_CFC_ (* Continuous Function Chart, elements in execution order *)
#0 MOVE(EN: SCHU_P2_4_RESET_DF_VALUE, SCHU_P2_4_M_MAXSPEED_df)
#1 SCHU_P2_4_M_MAXSPEED <= #0
#2 MOVE(EN: SCHU_P2_4_RESET_DF_VALUE, SCHU_P2_4_M_MINSPEED_df)
#3 SCHU_P2_4_M_MINSPEED <= #2
#4 MOVE(EN: SCHU_P2_4_RESET_DF_VALUE, SCHU_P2_4_YA2_ZADER_RAS_df)
#5 SCHU_P2_4_YA2_ZADER_RAS <= #4
#6 MOVE(EN: SCHU_P2_4_RESET_DF_VALUE, SCHU_P2_4_YA2_UST_RASSOG_df)
#7 SCHU_P2_4_YA2_UST_RASSOG <= #6
#8 MOVE(EN: SCHU_P2_4_RESET_DF_VALUE, SCHU_P2_4_YA2_ZAD_NEISP_df)
#9 SCHU_P2_4_YA2_ZAD_NEISP <= #8
#10 MOVE(EN: SCHU_P2_4_RESET_DF_VALUE, SCHU_P2_4_YA2_ZAD_NAGR_df)
#11 SCHU_P2_4_YA2_ZAD_NAGR <= #10
#12 MOVE(EN: SCHU_P2_4_RESET_DF_VALUE, SCHU_P2_4_YA3_ZADER_OTK_df)
#13 SCHU_P2_4_YA3_ZADER_OTK <= #12
#14 MOVE(EN: SCHU_P2_4_RESET_DF_VALUE, SCHU_P2_4_YA3_ZADER_RAS_df)
#15 SCHU_P2_4_YA3_ZADER_RAS <= #14
#16 MOVE(EN: SCHU_P2_4_RESET_DF_VALUE, SCHU_P2_4_YA3_UST_RAS_POL_df)
#17 SCHU_P2_4_YA3_UST_RAS_POL <= #16
#18 MOVE(EN: SCHU_P2_4_RESET_DF_VALUE, SCHU_P2_4_YA3_UST_RAS_TEMP_df)
#19 SCHU_P2_4_YA3_UST_RAS_TEMP <= #18
#20 MOVE(EN: SCHU_P2_4_RESET_DF_VALUE, SCHU_P2_4_YA4_ZADER_OTK_TEMP_df)
#21 SCHU_P2_4_YA4_ZADER_OTK_TEMP <= #20
#22 MOVE(EN: SCHU_P2_4_RESET_DF_VALUE, SCHU_P2_4_YA4_ZADER_OTK_df)
#23 SCHU_P2_4_YA4_ZADER_OTK <= #22
#24 MOVE(EN: SCHU_P2_4_RESET_DF_VALUE, SCHU_P2_4_YA4_UST_RAS_TEMP_df)
#25 SCHU_P2_4_YA4_UST_RAS_TEMP <= #24
#26 MOVE(EN: SCHU_P2_4_RESET_DF_VALUE, SCHU_P2_4_YA4_UST_RAS_POL_df)
#27 SCHU_P2_4_YA4_UST_RAS_POL <= #26
#28 MOVE(EN: SCHU_P2_4_RESET_DF_VALUE, SCHU_P2_4_YA2_KP_df)
#29 SCHU_P2_4_YA2_KP <= #28
#30 MOVE(EN: SCHU_P2_4_RESET_DF_VALUE, SCHU_P2_4_YA2_TI_df)
#31 SCHU_P2_4_YA2_TI <= #30
#32 MOVE(EN: SCHU_P2_4_RESET_DF_VALUE, SCHU_P2_4_YA2_TV_df)
#33 SCHU_P2_4_YA2_TV <= #32
#34 MOVE(EN: SCHU_P2_4_RESET_DF_VALUE, SCHU_P2_4_YA2_TD_df)
#35 SCHU_P2_4_YA2_TD <= #34
#36 MOVE(EN: SCHU_P2_4_RESET_DF_VALUE, SCHU_P2_4_YA3_KP_df)
#37 SCHU_P2_4_YA3_KP <= #36
#38 MOVE(EN: SCHU_P2_4_RESET_DF_VALUE, SCHU_P2_4_YA3_TI_df)
#39 SCHU_P2_4_YA3_TI <= #38
#40 MOVE(EN: SCHU_P2_4_RESET_DF_VALUE, SCHU_P2_4_YA3_TV_df)
#41 SCHU_P2_4_YA3_TV <= #40
#42 MOVE(EN: SCHU_P2_4_RESET_DF_VALUE, SCHU_P2_4_YA3_TD_df)
#43 SCHU_P2_4_YA3_TD <= #42
#44 MOVE(EN: SCHU_P2_4_RESET_DF_VALUE, SCHU_P2_4_YA4_KP_df)
#45 SCHU_P2_4_YA4_KP <= #44
#46 MOVE(EN: SCHU_P2_4_RESET_DF_VALUE, SCHU_P2_4_YA4_TI_df)
#47 SCHU_P2_4_YA4_TI <= #46
#48 MOVE(EN: SCHU_P2_4_RESET_DF_VALUE, SCHU_P2_4_YA4_TV_df)
#49 SCHU_P2_4_YA4_TV <= #48
#50 MOVE(EN: SCHU_P2_4_RESET_DF_VALUE, SCHU_P2_4_YA4_TD_df)
#51 SCHU_P2_4_YA4_TD <= #50
#52 MOVE(EN: SCHU_P2_4_RESET_DF_VALUE, SCHU_P2_4_PE_KP_df)
#53 SCHU_P2_4_PE_KP <= #52
#54 MOVE(EN: SCHU_P2_4_RESET_DF_VALUE, SCHU_P2_4_PE_TI_df)
#55 SCHU_P2_4_PE_TI <= #54
#56 MOVE(EN: SCHU_P2_4_RESET_DF_VALUE, SCHU_P2_4_PE_TV_df)
#57 SCHU_P2_4_PE_TV <= #56
#58 MOVE(EN: SCHU_P2_4_RESET_DF_VALUE, SCHU_P2_4_PE_TD_df)
#59 SCHU_P2_4_PE_TD <= #58
#60 MOVE(EN: SCHU_P2_4_RESET_DF_VALUE, SCHU_P2_4_PE_PID_VKL_df)
#61 SCHU_P2_4_PE_PID_VKL <= #60
#62 MOVE(EN: SCHU_P2_4_RESET_DF_VALUE, SCHU_P2_4_PE1_UST_df)
#63 SCHU_P2_4_PE1_UST <= #62
#64 MOVE(EN: SCHU_P2_4_RESET_DF_VALUE, SCHU_P2_4_TE2_UST_PROG_df)
#65 SCHU_P2_4_TE2_UST_PROG <= #64
#66 MOVE(EN: SCHU_P2_4_RESET_DF_VALUE, SCHU_P2_4_TE2_ZASCH_df)
#67 SCHU_P2_4_TE2_ZASCH <= #66
#68 MOVE(EN: SCHU_P2_4_RESET_DF_VALUE, SCHU_P2_4_TE2_ZASCH_DOB_df)
#69 SCHU_P2_4_TE2_ZASCH_DOB <= #68
#70 MOVE(EN: SCHU_P2_4_RESET_DF_VALUE, SCHU_P2_4_TE2_ZASCH_OTKL_df)
#71 SCHU_P2_4_TE2_ZASCH_OTKL <= #70
#72 MOVE(EN: SCHU_P2_4_RESET_DF_VALUE, SCHU_P2_4_YA2_UP_MIN_df)
#73 SCHU_P2_4_YA2_UP_MIN <= #72
#74 MOVE(EN: SCHU_P2_4_RESET_DF_VALUE, SCHU_P2_4_UE1_T_UST_df)
#75 SCHU_P2_4_UE1_T_UST <= #74
#76 MOVE(EN: SCHU_P2_4_RESET_DF_VALUE, SCHU_P2_4_UE2_T_UST_df)
#77 SCHU_P2_4_UE2_T_UST <= #76
#78 MOVE(EN: SCHU_P2_4_RESET_DF_VALUE, SCHU_P2_4_UE3_T_UST_df)
#79 SCHU_P2_4_UE3_T_UST <= #78
#80 MOVE(EN: SCHU_P2_4_RESET_DF_VALUE, SCHU_P2_4_UE2_VL_UST_OTKL_df)
#81 SCHU_P2_4_UE2_VL_UST_OTKL <= #80
#82 MOVE(EN: SCHU_P2_4_RESET_DF_VALUE, SCHU_P2_4_UE2_VL_UST_VKL_df)
#83 SCHU_P2_4_UE2_VL_UST_VKL <= #82
#84 MOVE(EN: SCHU_P2_4_RESET_DF_VALUE, SCHU_P2_4_UE3_VL_UST_OTKL_df)
#85 SCHU_P2_4_UE3_VL_UST_OTKL <= #84
#86 MOVE(EN: SCHU_P2_4_RESET_DF_VALUE, SCHU_P2_4_UE3_VL_UST_VKL_df)
#87 SCHU_P2_4_UE3_VL_UST_VKL <= #86
#88 MOVE(EN: SCHU_P2_4_RESET_DF_VALUE, SCHU_P2_4_UST_ZIMA_df)
#89 SCHU_P2_4_UST_ZIMA <= #88
#90 MOVE(EN: SCHU_P2_4_RESET_DF_VALUE, SCHU_P2_4_UST_LETO_df)
#91 SCHU_P2_4_UST_LETO <= #90
#92 MOVE(EN: SCHU_P2_4_RESET_DF_VALUE, SCHU_P2_4_UST_SEZ_ZIMA_df)
#93 SCHU_P2_4_UST_SEZ_ZIMA <= #92
#94 MOVE(EN: SCHU_P2_4_RESET_DF_VALUE, SCHU_P2_4_UST_SEZ_LETO_df)
#95 SCHU_P2_4_UST_SEZ_LETO <= #94
_END_CFC_
(* the same logic as Structured Text *)
IF SCHU_P2_4_RESET_DF_VALUE THEN SCHU_P2_4_M_MAXSPEED := SCHU_P2_4_M_MAXSPEED_df; END_IF;
IF SCHU_P2_4_RESET_DF_VALUE THEN SCHU_P2_4_M_MINSPEED := SCHU_P2_4_M_MINSPEED_df; END_IF;
IF SCHU_P2_4_RESET_DF_VALUE THEN SCHU_P2_4_YA2_ZADER_RAS := SCHU_P2_4_YA2_ZADER_RAS_df; END_IF;
IF SCHU_P2_4_RESET_DF_VALUE THEN SCHU_P2_4_YA2_UST_RASSOG := SCHU_P2_4_YA2_UST_RASSOG_df; END_IF;
IF SCHU_P2_4_RESET_DF_VALUE THEN SCHU_P2_4_YA2_ZAD_NEISP := SCHU_P2_4_YA2_ZAD_NEISP_df; END_IF;
IF SCHU_P2_4_RESET_DF_VALUE THEN SCHU_P2_4_YA2_ZAD_NAGR := SCHU_P2_4_YA2_ZAD_NAGR_df; END_IF;
IF SCHU_P2_4_RESET_DF_VALUE THEN SCHU_P2_4_YA3_ZADER_OTK := SCHU_P2_4_YA3_ZADER_OTK_df; END_IF;
IF SCHU_P2_4_RESET_DF_VALUE THEN SCHU_P2_4_YA3_ZADER_RAS := SCHU_P2_4_YA3_ZADER_RAS_df; END_IF;
IF SCHU_P2_4_RESET_DF_VALUE THEN SCHU_P2_4_YA3_UST_RAS_POL := SCHU_P2_4_YA3_UST_RAS_POL_df; END_IF;
IF SCHU_P2_4_RESET_DF_VALUE THEN SCHU_P2_4_YA3_UST_RAS_TEMP := SCHU_P2_4_YA3_UST_RAS_TEMP_df; END_IF;
IF SCHU_P2_4_RESET_DF_VALUE THEN SCHU_P2_4_YA4_ZADER_OTK_TEMP := SCHU_P2_4_YA4_ZADER_OTK_TEMP_df; END_IF;
IF SCHU_P2_4_RESET_DF_VALUE THEN SCHU_P2_4_YA4_ZADER_OTK := SCHU_P2_4_YA4_ZADER_OTK_df; END_IF;
IF SCHU_P2_4_RESET_DF_VALUE THEN SCHU_P2_4_YA4_UST_RAS_TEMP := SCHU_P2_4_YA4_UST_RAS_TEMP_df; END_IF;
IF SCHU_P2_4_RESET_DF_VALUE THEN SCHU_P2_4_YA4_UST_RAS_POL := SCHU_P2_4_YA4_UST_RAS_POL_df; END_IF;
IF SCHU_P2_4_RESET_DF_VALUE THEN SCHU_P2_4_YA2_KP := SCHU_P2_4_YA2_KP_df; END_IF;
IF SCHU_P2_4_RESET_DF_VALUE THEN SCHU_P2_4_YA2_TI := SCHU_P2_4_YA2_TI_df; END_IF;
IF SCHU_P2_4_RESET_DF_VALUE THEN SCHU_P2_4_YA2_TV := SCHU_P2_4_YA2_TV_df; END_IF;
IF SCHU_P2_4_RESET_DF_VALUE THEN SCHU_P2_4_YA2_TD := SCHU_P2_4_YA2_TD_df; END_IF;
IF SCHU_P2_4_RESET_DF_VALUE THEN SCHU_P2_4_YA3_KP := SCHU_P2_4_YA3_KP_df; END_IF;
IF SCHU_P2_4_RESET_DF_VALUE THEN SCHU_P2_4_YA3_TI := SCHU_P2_4_YA3_TI_df; END_IF;
IF SCHU_P2_4_RESET_DF_VALUE THEN SCHU_P2_4_YA3_TV := SCHU_P2_4_YA3_TV_df; END_IF;
IF SCHU_P2_4_RESET_DF_VALUE THEN SCHU_P2_4_YA3_TD := SCHU_P2_4_YA3_TD_df; END_IF;
IF SCHU_P2_4_RESET_DF_VALUE THEN SCHU_P2_4_YA4_KP := SCHU_P2_4_YA4_KP_df; END_IF;
IF SCHU_P2_4_RESET_DF_VALUE THEN SCHU_P2_4_YA4_TI := SCHU_P2_4_YA4_TI_df; END_IF;
IF SCHU_P2_4_RESET_DF_VALUE THEN SCHU_P2_4_YA4_TV := SCHU_P2_4_YA4_TV_df; END_IF;
IF SCHU_P2_4_RESET_DF_VALUE THEN SCHU_P2_4_YA4_TD := SCHU_P2_4_YA4_TD_df; END_IF;
IF SCHU_P2_4_RESET_DF_VALUE THEN SCHU_P2_4_PE_KP := SCHU_P2_4_PE_KP_df; END_IF;
IF SCHU_P2_4_RESET_DF_VALUE THEN SCHU_P2_4_PE_TI := SCHU_P2_4_PE_TI_df; END_IF;
IF SCHU_P2_4_RESET_DF_VALUE THEN SCHU_P2_4_PE_TV := SCHU_P2_4_PE_TV_df; END_IF;
IF SCHU_P2_4_RESET_DF_VALUE THEN SCHU_P2_4_PE_TD := SCHU_P2_4_PE_TD_df; END_IF;
IF SCHU_P2_4_RESET_DF_VALUE THEN SCHU_P2_4_PE_PID_VKL := SCHU_P2_4_PE_PID_VKL_df; END_IF;
IF SCHU_P2_4_RESET_DF_VALUE THEN SCHU_P2_4_PE1_UST := SCHU_P2_4_PE1_UST_df; END_IF;
IF SCHU_P2_4_RESET_DF_VALUE THEN SCHU_P2_4_TE2_UST_PROG := SCHU_P2_4_TE2_UST_PROG_df; END_IF;
IF SCHU_P2_4_RESET_DF_VALUE THEN SCHU_P2_4_TE2_ZASCH := SCHU_P2_4_TE2_ZASCH_df; END_IF;
IF SCHU_P2_4_RESET_DF_VALUE THEN SCHU_P2_4_TE2_ZASCH_DOB := SCHU_P2_4_TE2_ZASCH_DOB_df; END_IF;
IF SCHU_P2_4_RESET_DF_VALUE THEN SCHU_P2_4_TE2_ZASCH_OTKL := SCHU_P2_4_TE2_ZASCH_OTKL_df; END_IF;
IF SCHU_P2_4_RESET_DF_VALUE THEN SCHU_P2_4_YA2_UP_MIN := SCHU_P2_4_YA2_UP_MIN_df; END_IF;
IF SCHU_P2_4_RESET_DF_VALUE THEN SCHU_P2_4_UE1_T_UST := SCHU_P2_4_UE1_T_UST_df; END_IF;
IF SCHU_P2_4_RESET_DF_VALUE THEN SCHU_P2_4_UE2_T_UST := SCHU_P2_4_UE2_T_UST_df; END_IF;
IF SCHU_P2_4_RESET_DF_VALUE THEN SCHU_P2_4_UE3_T_UST := SCHU_P2_4_UE3_T_UST_df; END_IF;
IF SCHU_P2_4_RESET_DF_VALUE THEN SCHU_P2_4_UE2_VL_UST_OTKL := SCHU_P2_4_UE2_VL_UST_OTKL_df; END_IF;
IF SCHU_P2_4_RESET_DF_VALUE THEN SCHU_P2_4_UE2_VL_UST_VKL := SCHU_P2_4_UE2_VL_UST_VKL_df; END_IF;
IF SCHU_P2_4_RESET_DF_VALUE THEN SCHU_P2_4_UE3_VL_UST_OTKL := SCHU_P2_4_UE3_VL_UST_OTKL_df; END_IF;
IF SCHU_P2_4_RESET_DF_VALUE THEN SCHU_P2_4_UE3_VL_UST_VKL := SCHU_P2_4_UE3_VL_UST_VKL_df; END_IF;
IF SCHU_P2_4_RESET_DF_VALUE THEN SCHU_P2_4_UST_ZIMA := SCHU_P2_4_UST_ZIMA_df; END_IF;
IF SCHU_P2_4_RESET_DF_VALUE THEN SCHU_P2_4_UST_LETO := SCHU_P2_4_UST_LETO_df; END_IF;
IF SCHU_P2_4_RESET_DF_VALUE THEN SCHU_P2_4_UST_SEZ_ZIMA := SCHU_P2_4_UST_SEZ_ZIMA_df; END_IF;
IF SCHU_P2_4_RESET_DF_VALUE THEN SCHU_P2_4_UST_SEZ_LETO := SCHU_P2_4_UST_SEZ_LETO_df; END_IF;
END_PROGRAM

(* POU Persist, ST *)
PROGRAM Persist
VAR
	Save: WritePersistentData;
END_VAR
Save(NETID:='10.150.4.76.1.1',PORT:=801,START:=TRUE,TMOUT:=t#1s ,BUSY=> ,ERR=> ,	ERRID=> );
Save(NETID:='10.150.4.76.1.1',PORT:=801,START:= FALSE ,TMOUT:=t#1s ,BUSY=> ,ERR=> ,ERRID=> );
END_PROGRAM

(* POU Input/ALL_Input, CFC *)
PROGRAM ALL_Input
VAR
END_VAR
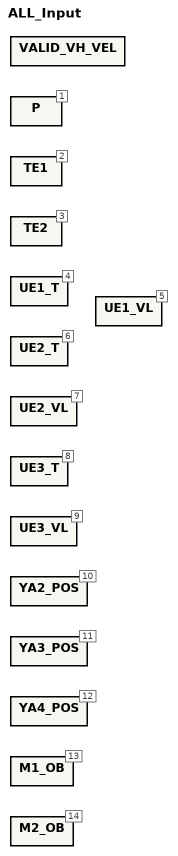
_CFC_ (* Continuous Function Chart, elements in execution order *)
#0 VALID_VH_VEL()
#1 P()
#2 TE1()
#3 TE2()
#4 UE1_T()
#5 UE1_VL()
#6 UE2_T()
#7 UE2_VL()
#8 UE3_T()
#9 UE3_VL()
#10 YA2_POS()
#11 YA3_POS()
#12 YA4_POS()
#13 M1_OB()
#14 M2_OB()
_END_CFC_
(* the same logic as Structured Text *)
VALID_VH_VEL();
P();
TE1();
TE2();
UE1_T();
UE1_VL();
UE2_T();
UE2_VL();
UE3_T();
UE3_VL();
YA2_POS();
YA3_POS();
YA4_POS();
M1_OB();
M2_OB();
END_PROGRAM

(* POU Input/VALID_VH_VEL, CFC *)
PROGRAM VALID_VH_VEL
VAR
	SCHU_P2_4_UST_SEZ_LETO_OLD: REAL;
	SCHU_P2_4_UST_SEZ_ZIMA_OLD: REAL;

	RT_VKL_OLD_SEZ_LETO: R_TRIG;
	RT_VKL_OLD_SEZ_ZIMA: R_TRIG;

	(*_____________________________________*)
	SCHU_P2_4_UE2_VL_UST_OTKL_OLD: REAL;
	SCHU_P2_4_UE2_VL_UST_VKL_OLD: REAL;

	RT_UE2_VL_UST_OTKL_OLD: R_TRIG;
	RT_UE2_VL_UST_VKL_OLD: R_TRIG;

	(*_____________________________________*)
	RT_UE3_VL_UST_OTKL_OLD: R_TRIG;
	RT_UE3_VL_UST_VKL_OLD: R_TRIG;
	SCHU_P2_4_UE3_VL_UST_OTKL_OLD: REAL;
	SCHU_P2_4_UE3_VL_UST_VKL_OLD: REAL;

	(*_____________________________________*)
	RT_UE2_TE_UST_OTKL_OLD: R_TRIG;
	RT_UE3_TE_UST_VKL_OLD: R_TRIG;

	SCHU_P2_4_UE1_T_UST_OLD: REAL;
	SCHU_P2_4_UE2_T_UST_OLD: REAL;
	SCHU_P2_4_UE3_T_UST_OLD: REAL;
END_VAR
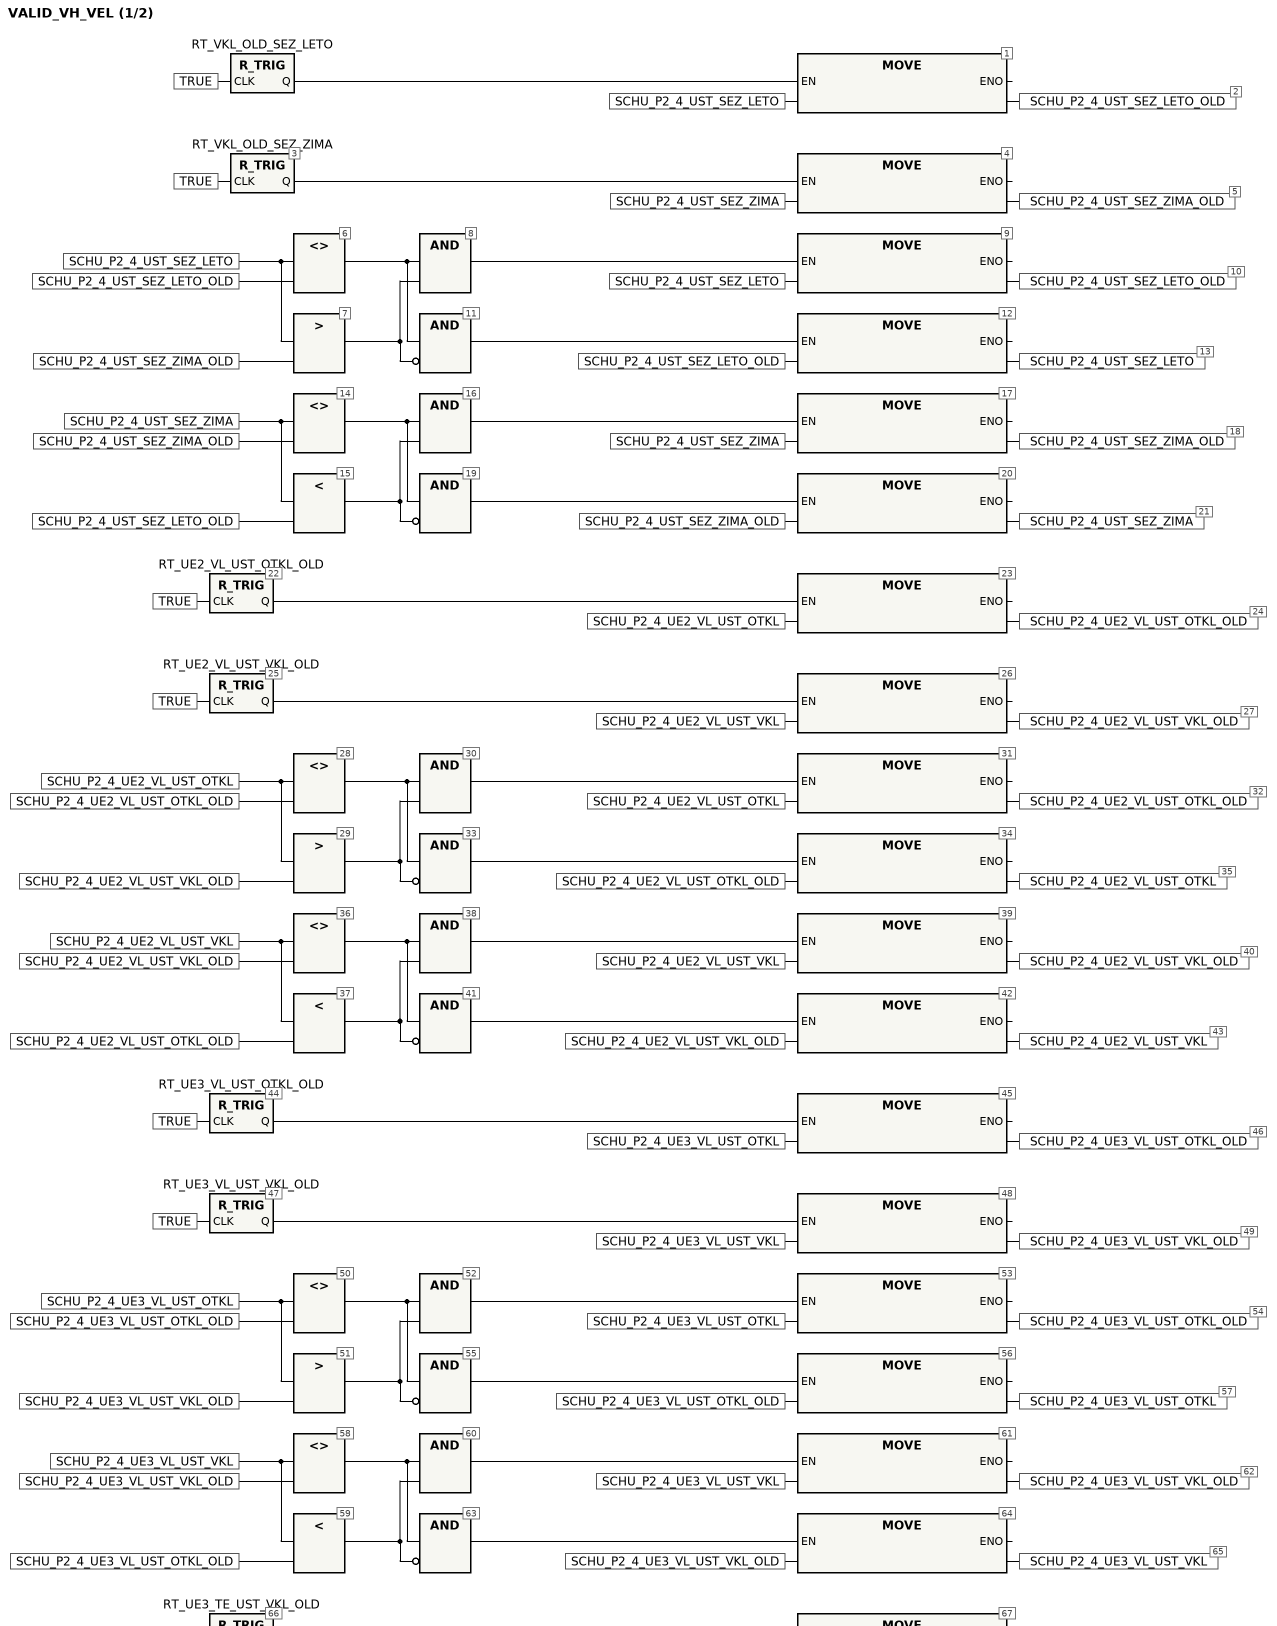
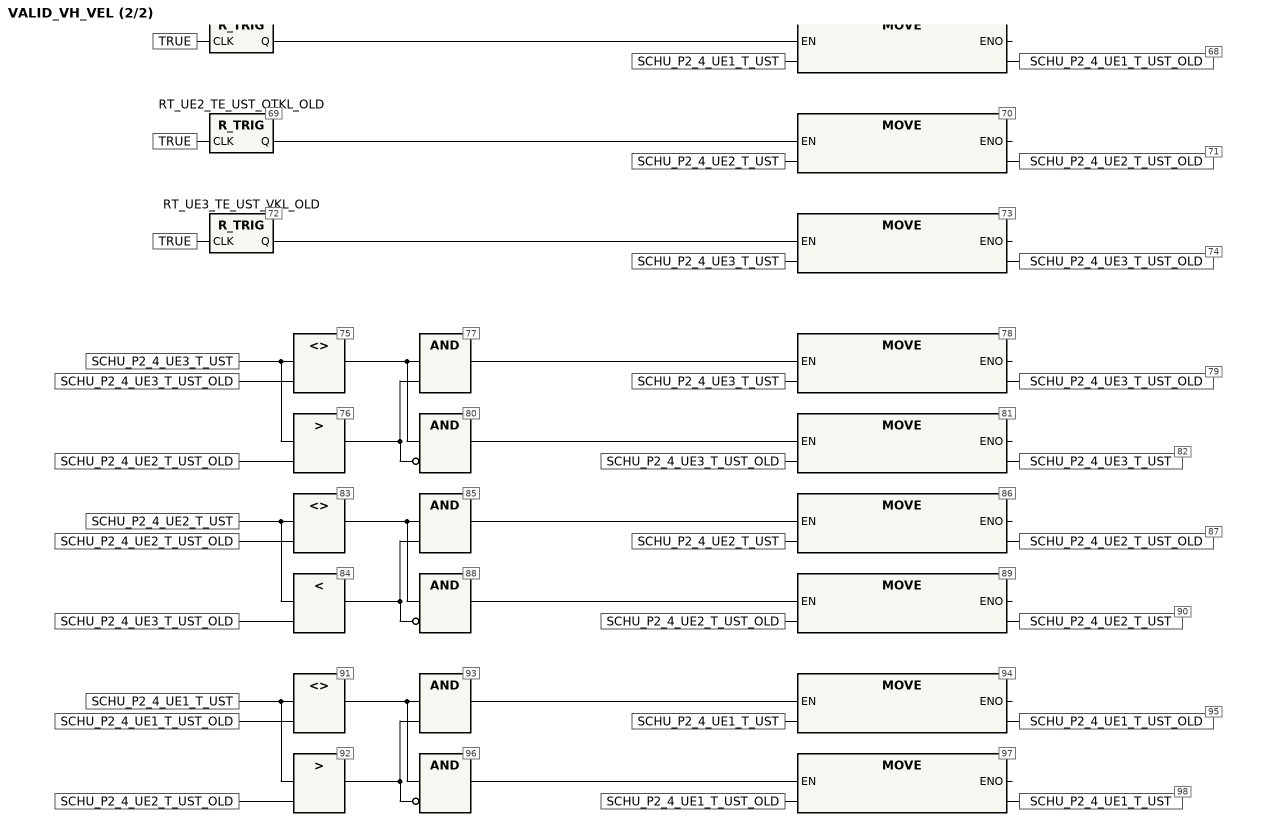
